// TIA Portal V16 export
// export: Created 2021-07-12T14:47:20.2714515Z, ExportSetting WithDefaults, DisplayName Totally Integrated Automation Portal, DisplayVersion V16, DisplayName TIA Portal Version Control Interface, DisplayVersion V16, DisplayName TIA Portal Openness, DisplayVersion V16, DisplayName STEP 7 Professional, DisplayVersion V16, DisplayName STEP 7 Safety, DisplayVersion V16, DisplayName WinCC Professional, DisplayVersion V16
TYPE "SimaHydTO_typeHMIConnectionAxisSelector"
TITLE = SimaHydTO_typeHMIConnectionAxisSelector
// HMI interface: Axis selection of axis array
// stored: IsFailsafeCompliant false
   STRUCT
      Command { S7_SetPoint := 'True'} : "SimaHydTO_typeHMIConnectionAxisSelectorCommand";   // Data: HMI -> PLC
      Status { S7_SetPoint := 'True'} : "SimaHydTO_typeHMIConnectionAxisSelectorStatus";   // Data: PLC -> HMI
   END_STRUCT;
END_TYPE
